(* IEC 61131-3 sources: CodesysTest/alpha/export/FBs/Components/Motors/Applied Motion/FB_AppliedMotionStepServoEIPPassthrough_1.pou, 2 files *)

(* ---- FB_AppliedMotionStepServoEIPPassthrough_1.pou.st ---- *)
(*#-#-#-#-#-#-#-#-#-#---Declaration---#-#-#-#-#-#-#-#-#-#-#-#-#*)

FUNCTION_BLOCK FB_AppliedMotionStepServoEIPPassthrough_1 EXTENDS FB_AppliedMotionStepServoEIPPassthrough
VAR_INPUT
END_VAR
VAR_OUTPUT
END_VAR
VAR
END_VAR
(*#-#-#-#-#-#-#-#-#-#---Implementation---#-#-#-#-#-#-#-#-#-#-#-#-#*)

SUPER^();

(* ---- AllowClamping.m.st ---- *)
(*#-#-#-#-#-#-#-#-#-#---Declaration---#-#-#-#-#-#-#-#-#-#-#-#-#*)

METHOD AllowClamping
VAR_INPUT
END_VAR
(*#-#-#-#-#-#-#-#-#-#---Implementation---#-#-#-#-#-#-#-#-#-#-#-#-#*)

MoveDistanceTorque(velocity:=100, acceleration := 1, deceleration := 1, distance := 0, current := 1);
